INTERFACE I_File

// close file
METHOD PUBLIC M_Close : BOOL
VAR_INPUT
END_VAR
END_METHOD

// Delete file
METHOD PUBLIC M_Delete : BOOL
VAR_INPUT
    sFileName : STRING(255);
END_VAR
END_METHOD

// get file size
METHOD PUBLIC M_GetSize : UDINT
VAR_INPUT
END_VAR
END_METHOD

// Open file
METHOD PUBLIC M_Open : BOOL
VAR_INPUT
    sFileName:				STRING(255);
	eMode: 					SysFile.ACCESS_MODE := SysFile.AM_APPEND_PLUS;
END_VAR
END_METHOD

// Read file
METHOD PUBLIC M_Read : BOOL
VAR_INPUT
END_VAR
END_METHOD

// state of file
METHOD PUBLIC M_Status : E_FileState
VAR_INPUT
END_VAR
END_METHOD

// Write file
METHOD PUBLIC M_Write : BOOL
VAR_INPUT
	pBuffer:	POINTER TO BYTE;
    nSize:     	UDINT;
END_VAR
END_METHOD

END_INTERFACE

(* stored: Version 1.1.0.1
   Itf I_File: Id {0398998b-406f-4dc3-884a-bd60146ff034}
   Method M_Close: Id {81246933-abb8-43ee-80a3-7db556a2806f}
   Method M_Delete: Id {1ab6a5d3-e618-451b-9a6d-bf65e2d28017}
   Method M_GetSize: Id {4536dbc1-2529-4d82-83a4-0005239e6472}
   Method M_Open: Id {c3646e36-af69-41b6-8691-3fff7524229e}
   Method M_Read: Id {c1c6e01c-368e-48e5-b6be-1ea452c44e04}
   Method M_Status: Id {7d1bdc79-1243-4e4d-a54a-8b2b8fe5d17b}
   Method M_Write: Id {5ca68eff-0689-40be-acb5-491e1faac60d} *)
